// TIA Portal V18 export
TYPE "KISTLER_TO_PLC"
// stored: IsFailsafeCompliant false
   STRUCT
      "0.0" : Bool;   // Mirrored cycle start
      "0.1" : Bool;   // Mirrored Channel Y (Force) Tare Or Reset Piezo
      "0.2" : Bool;   // Mirrored Channel X (Position) Reset
      "0.3" : Bool;   // Mirrored Trigger Sensor Test For X
      "0.4" : Bool;   // Mirrored Trigger Sensor Test For Y
      "0.5" : Bool;
      "0.6" : Bool;   // Mirrored master measurement
      "0.7" : Bool;   // Mirrored Zero Incremental Encoder
      "1.0" : Bool;
      "1.1" : Bool;   // Mirrored Acknowledgement With Admin Rights
      "1.2" : Bool;
      "1.3" : Bool;   // Mirrored ACCESS
      "1.4" : Bool;   // Mirrored production mode
      "1.5" : Bool;   // Mirrored Reset Statistics
      "1.6" : Bool;   // Mirrored Deactivate Statistics
      "1.7" : Bool;   // Mirrored Ext. channel Y Tare or Reset Piezo (MaXYmos NC)
      "2" : Byte;   // Mirrored Measurement program selection
      "3.0" : Bool;   // Reserved
      "3.1" : Bool;   // Reserved
      "3.2" : Bool;   // Mirrored resetting of global serial number
      "3.3" : Bool;   // Reserved
      "3.4" : Bool;   // Reserved
      "3.5" : Bool;   // Brake test is performed
      "3.6" : Bool;   // Reserved
      "3.7" : Bool;   // Reserved
      "4.0" : Bool;   // UNI_0
      "4.1" : Bool;   // UNI_1
      "4.2" : Bool;   // UNI_2
      "4.3" : Bool;   // UNI_3
      "4.4" : Bool;   // UNI_4
      "4.5" : Bool;   // UNI_5
      "4.6" : Bool;   // UNI_6
      "4.7" : Bool;   // UNI_7
      "5.0" : Bool;   // Reserved
      "5.1" : Bool;   // Reserved
      "5.2" : Bool;   // Reserved
      "5.3" : Bool;   // Reserved
      "5.4" : Bool;   // Reserved
      "5.5" : Bool;   // Reserved
      "5.6" : Bool;   // Reserved
      "5.7" : Bool;   // Reserved
      "6.0" : Bool;   // Already
      "6.1" : Bool;   // Result GOOD
      "6.2" : Bool;   // Result BAD
      "6.3" : Bool;   // No pass exceeded
      "6.4" : Bool;   // Reserved
      "6.5" : Bool;   // Reserved
      "6.6" : Bool;   // Warning
      "6.7" : Bool;   // Alarm
      "7.0" : Bool;   // Swichting signal S1
      "7.1" : Bool;   // Swichting signal S2
      "7.2" : Bool;   // Reserved
      "7.3" : Bool;   // Reserved
      "7.4" : Bool;   // Reserved
      "7.5" : Bool;   // Reserved
      "7.6" : Bool;   // Reserved
      "7.7" : Bool;   // Reserved
      "8.0" : Bool;   // UNI_0（Freely configurable digital Output signal）
      "8.1" : Bool;   // UNI_1
      "8.2" : Bool;   // UNI_2
      "8.3" : Bool;   // UNI_3
      "8.4" : Bool;   // UNI_4
      "8.5" : Bool;   // UNI_5
      "8.6" : Bool;   // UNI_6
      "8.7" : Bool;   // UNI_7
      "9.0" : Bool;   // Mirrored Enable Drive
      "9.1" : Bool;   // Mirrored Command process of the sequence
      "9.2" : Bool;   // Mirrored Command movement to home position (MP-specific)
      "9.3" : Bool;   // Mirrored Command movement to reference position (global)
      "9.4" : Bool;   // Mirrored Command jogging forwards
      "9.5" : Bool;   // Mirrored Command jogging Backwards
      "9.6" : Bool;   // Output is set through sequence object Wait. Sequence wants it for continue
      "9.7" : Bool;   // Brake Test Is Performed
      "10.0" : Bool;   // Sequence/command Stopped
      "10.1" : Bool;   // Sequence/command ended
      "10.2" : Bool;   // NOK for online evaluation of a corresponding EOs.
      "10.3" : Bool;   // External stop was set in sequence object
      "10.4" : Bool;   // Sequence/command error
      "10.5" : Bool;   // Enable drive set (current status of the enable)
      "10.6" : Bool;   // Home position reached (NC joining module is in MP-specific home pos)
      "10.7" : Bool;   // Reference position reached (NC joining module is in global reference position)
      "11.0" : Bool;   // StandStill
      "11.1" : Bool;   // Brake test required
      "11.2" : Bool;   // Warning message on the servo amplifier pending
      "11.3" : Bool;   // Alarm message on the servo amplifier pending
      "11.4" : Bool;   // Safety Status SMES Active
      "11.5" : Bool;   // Safety Status SMST2 Active
      "11.6" : Bool;   // Safety Status SMM1 Active
      "11.7" : Bool;   // 1= Service Mode By Kistler Panel Is Active
      "12.0" : Bool;   // Mirrored Select sequence main, Sub1 ... 3
      "12.1" : Bool;   // Mirrored Select sequence main, Sub1 ... 3
      "12.2" : Bool;   // Reserved
      "12.3" : Bool;   // Reserved
      "12.4" : Bool;   // Reserved
      "12.5" : Bool;   // Reserved
      "12.6" : Bool;   // Reserved
      "12.7" : Bool;   // Reserved
      "13" : Byte;   // Labear 2
      "14" : Byte;   // Mirrored measurement program choice of the input telegram
      "15.0" : Bool;   // Reserved
      "15.1" : Bool;   // Reserved
      "15.2" : Bool;   // Reserved
      "15.3" : Bool;   // Reserved
      "15.4" : Bool;   // Reserved
      "15.5" : Bool;   // Reserved
      "15.6" : Bool;   // Reserved
      "15.7" : Bool;   // If bit is set, the telegram data are interpreted as a global object
      "16" : Byte;   // Mirror CFG-ADR
      "17" : Byte;   // Mirror CFG-LENGHT
      "18.0" : Bool;   // Mirror Select-page
      "18.1" : Bool;   // Mirror Select-page
      "18.2" : Bool;   // Mirror Select-page
      "18.3" : Bool;   // Reserved
      "18.4" : Bool;   // Reserved
      "18.5" : Bool;   // Reserved
      "18.6" : Bool;   // Reserved
      "18.7" : Bool;   // Reserved
      "19.0" : Bool;   // Trasmission fault
      "19.1" : Bool;   // Ack
      "19.2" : Bool;   // Device available
      "19.3" : Bool;   // Reserved
      "19.4" : Bool;   // Selected Map
      "19.5" : Bool;   // Reserved
      "19.6" : Bool;   // Global
      "19.7" : Bool;   // Backup request
      "20" : Real;   // Force actual [kN]
      "24" : Real;   // Position actual [mm]
      "28" : Real;   // Max press force [kN]
      "32" : Real;   // Final distance [mm]
      "36" : Real;   // Position actual [mm]1
      EO_01 : Struct
         MaxForceCurPoS : Real;
         MaxForce : Real;
      END_STRUCT;
      EO_02 : Struct
         MaxForceCurPoS : Real;
         MaxForce : Real;
      END_STRUCT;
      EO_03 : Struct
         MaxForceCurPoS : Real;
         MaxForce : Real;
      END_STRUCT;
      EO_04 : Struct
         MaxForceCurPoS : Real;
         MaxForce : Real;
      END_STRUCT;
      EO_05 : Struct
         MaxForceCurPoS : Real;
         MaxForce : Real;
      END_STRUCT;
      EO_06 : Struct
         MaxForceCurPoS : Real;
         MaxForce : Real;
      END_STRUCT;
      "88" : Byte;   // pvEolastResult1(1:OK 2:NG)
      "89" : Byte;   // pvEolastResult2(1:OK 2:NG)
      "90" : Byte;   // pvEolastResult3(1:OK 2:NG)
      "91" : Byte;   // pvEolastResult4(1:OK 2:NG)
      "92" : Byte;   // pvEolastResult5(1:OK 2:NG)
      "93" : Byte;   // pvEolastResult6(1:OK 2:NG)
      "94" : Array[1..126] of Byte;
   END_STRUCT;
END_TYPE
